// TIA Portal V20 export
DATA_BLOCK "Data_block_1"   // DB5
// stored: Access Published, MemoryReserve 100, Namespace ELY_1
   VAR
      process_done : Bool;
   END_VAR
BEGIN
END_DATA_BLOCK
